// LS Electric XG5000 project: 16-39-1
// PLC NewPLC
// module base 0 slot 0: 입출력 모듈:XBC-DR14E (DC 24V 입력 8점, 릴레이 출력 6점)

PROGRAM NewProgram (task: 스캔 프로그램)

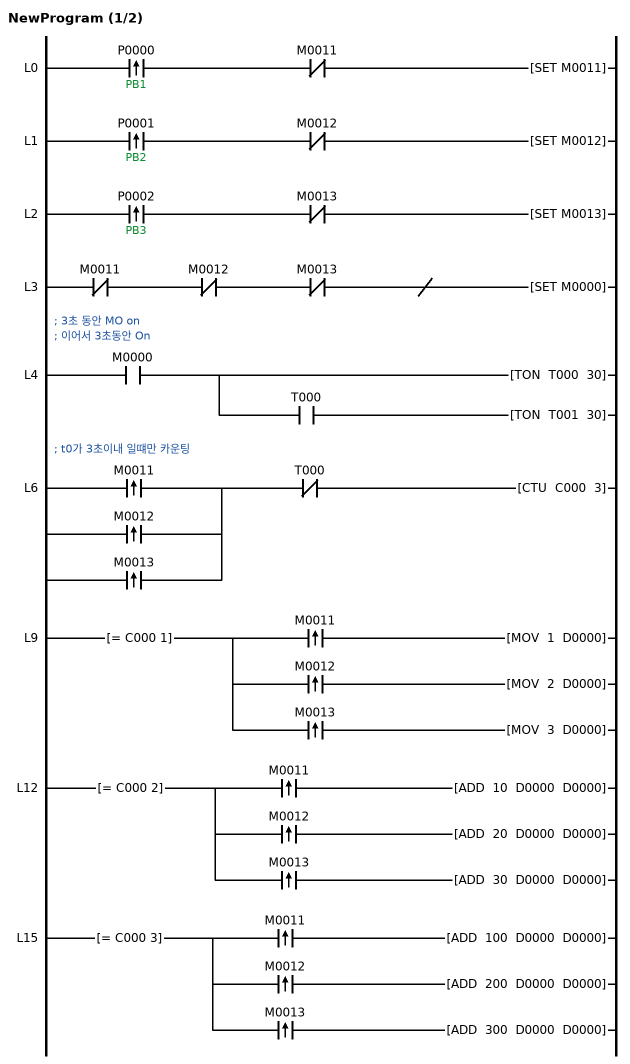
; L0
LOADP     P0000	// PB1
AND NOT   M0011
SET       M0011
; L1
LOADP     P0001	// PB2
AND NOT   M0012
SET       M0012
; L2
LOADP     P0002	// PB3
AND NOT   M0013
SET       M0013
; L3
LOAD NOT  M0011
AND NOT   M0012
AND NOT   M0013
NOT
SET       M0000
; L4
LOAD      M0000
TON       T000 30
AND       T000
TON       T001 30
// output comment: 3초 동안 MO on
// output comment: 이어서 3초동안 On
; L6
LOADP     M0011
ORP       M0012
ORP       M0013
AND NOT   T000
CTU       C000 3
// output comment: t0가 3초이내 일떄만 카운팅
; L9
LOAD=     C000 1
MPUSH
ANDP      M0011
MOV       1 D0000
MLOAD
ANDP      M0012
MOV       2 D0000
MPOP
ANDP      M0013
MOV       3 D0000
; L12
LOAD=     C000 2
MPUSH
ANDP      M0011
ADD       10 D0000 D0000
MLOAD
ANDP      M0012
ADD       20 D0000 D0000
MPOP
ANDP      M0013
ADD       30 D0000 D0000
; L15
LOAD=     C000 3
MPUSH
ANDP      M0011
ADD       100 D0000 D0000
MLOAD
ANDP      M0012
ADD       200 D0000 D0000
MPOP
ANDP      M0013
ADD       300 D0000 D0000

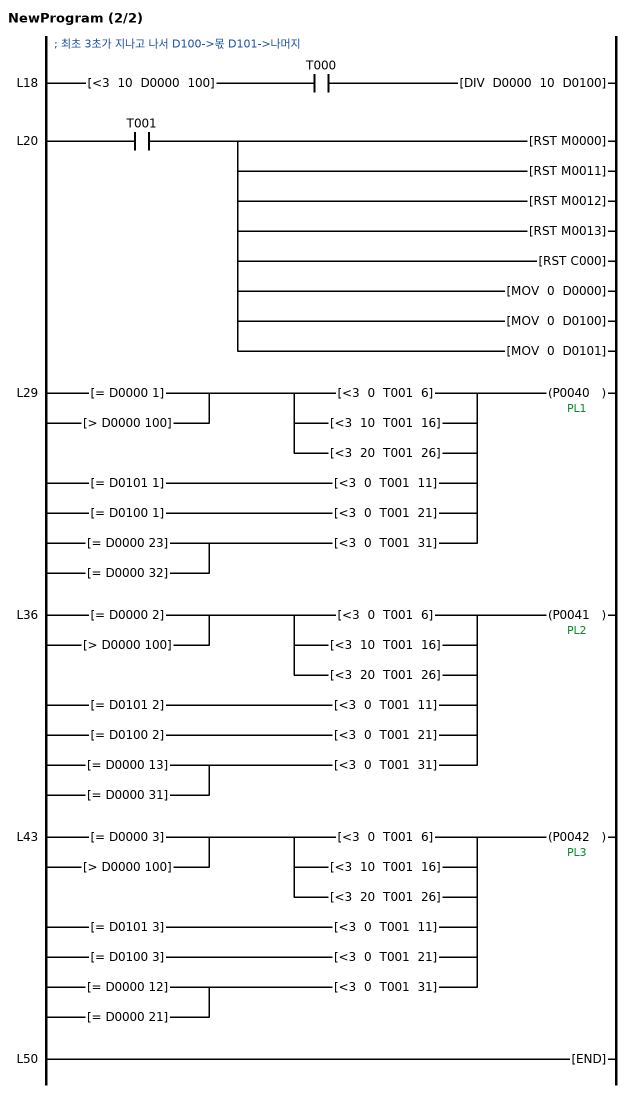
; L18
LOAD<3    10 D0000 100
AND       T000
DIV       D0000 10 D0100
// output comment: 최초 3초가 지나고 나서 D100->몫 D101->나머지
; L20
LOAD      T001
RST       M0000
RST       M0011
RST       M0012
RST       M0013
RST       C000
MOV       0 D0000
MOV       0 D0100
MOV       0 D0101
; L29
LOAD=     D0000 1
OR>       D0000 100
LOAD<3    0 T001 6
OR<3      10 T001 16
OR<3      20 T001 26
AND LOAD
LOAD=     D0101 1
AND<3     0 T001 11
OR LOAD
LOAD=     D0100 1
AND<3     0 T001 21
OR LOAD
LOAD=     D0000 23
OR=       D0000 32
AND<3     0 T001 31
OR LOAD
OUT       P0040	// PL1
; L36
LOAD=     D0000 2
OR>       D0000 100
LOAD<3    0 T001 6
OR<3      10 T001 16
OR<3      20 T001 26
AND LOAD
LOAD=     D0101 2
AND<3     0 T001 11
OR LOAD
LOAD=     D0100 2
AND<3     0 T001 21
OR LOAD
LOAD=     D0000 13
OR=       D0000 31
AND<3     0 T001 31
OR LOAD
OUT       P0041	// PL2
; L43
LOAD=     D0000 3
OR>       D0000 100
LOAD<3    0 T001 6
OR<3      10 T001 16
OR<3      20 T001 26
AND LOAD
LOAD=     D0101 3
AND<3     0 T001 11
OR LOAD
LOAD=     D0100 3
AND<3     0 T001 21
OR LOAD
LOAD=     D0000 12
OR=       D0000 21
AND<3     0 T001 31
OR LOAD
OUT       P0042	// PL3
; L50
END